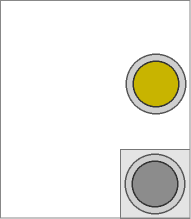
VISUALIZATION VisualizationSquareWaveGenerator  // 191x219
    PushSwitch (120,149 70x70), behaviour: TOGGLE, style: Switch-PushSwitch-Gray
    Lamp1 (121,49 70x70), variable: MAIN.bPulse, style: Lamp-Lamp1-Yellow
END_VISUALIZATION

(* stored: Version 1.1.0.1, ProductVersion 3.1.4024.12
   Visu VisualizationSquareWaveGenerator: Id {e1a1e3dc-cc93-48f0-9edc-d03367f237f4} *)
